FUNCTION_BLOCK IO_RouteAI (* Backend router for IO_AI: 0 simulated, 1 GPIO, 2 Modbus *)
  (* Standard: 61499-2 *)
  (* Version 0.1, 2026-09-28, Project contributors, AAU Smart Production Lab *)
  PACKAGE unitlib;
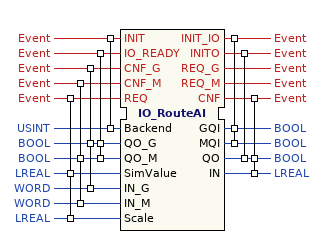
  EVENT_INPUT
    INIT WITH Backend;
    IO_READY WITH QO_G, QO_M;
    CNF_G WITH QO_G, IN_G;
    CNF_M WITH QO_M, IN_M;
    REQ WITH SimValue, Scale;
  END_EVENT
  EVENT_OUTPUT
    INIT_IO WITH GQI, MQI;
    INITO WITH QO;
    REQ_G;
    REQ_M;
    CNF WITH QO, IN;
  END_EVENT
  VAR_INPUT
    Backend : USINT;
    QO_G : BOOL;
    QO_M : BOOL;
    SimValue : LREAL;
    IN_G : WORD;
    IN_M : WORD;
    Scale : LREAL := 1.0;
  END_VAR
  VAR_OUTPUT
    GQI : BOOL;
    MQI : BOOL;
    QO : BOOL;
    IN : LREAL;
  END_VAR
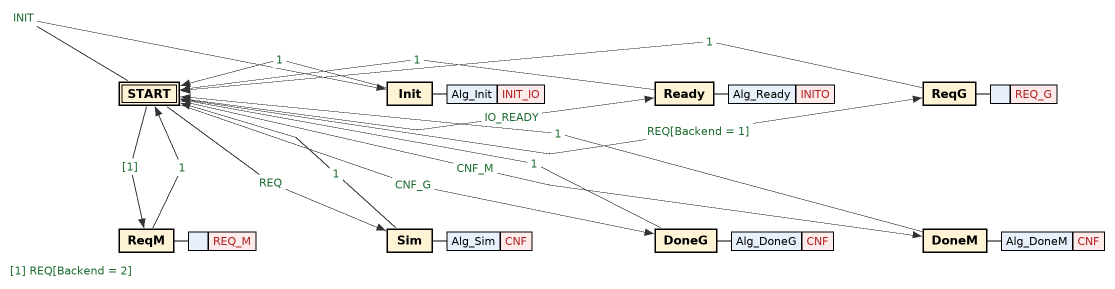
  EC_STATES
    START;
    Init : Alg_Init -> INIT_IO;
    Ready : Alg_Ready -> INITO;
    ReqG : -> REQ_G;
    ReqM : -> REQ_M;
    Sim : Alg_Sim -> CNF;
    DoneG : Alg_DoneG -> CNF;
    DoneM : Alg_DoneM -> CNF;
  END_STATES
  EC_TRANSITIONS
    START TO Init := INIT;
    Init TO START := 1;
    START TO Ready := IO_READY;
    Ready TO START := 1;
    START TO ReqG := REQ[Backend = 1];
    START TO ReqM := REQ[Backend = 2];
    START TO Sim := REQ;
    START TO DoneG := CNF_G;
    START TO DoneM := CNF_M;
    ReqG TO START := 1;
    ReqM TO START := 1;
    Sim TO START := 1;
    DoneG TO START := 1;
    DoneM TO START := 1;
  END_TRANSITIONS
  ALGORITHM Alg_Init IN ST:
GQI := Backend = 1;
MQI := Backend = 2;
  END_ALGORITHM
  ALGORITHM Alg_Ready IN ST:
QO := (Backend = 0) OR ((Backend = 1) AND QO_G) OR ((Backend = 2) AND QO_M);
  END_ALGORITHM
  ALGORITHM Alg_Sim IN ST:
QO := TRUE;
IN := SimValue;
  END_ALGORITHM
  ALGORITHM Alg_DoneG IN ST:
QO := QO_G;
IN := UINT_TO_LREAL(WORD_TO_UINT(IN_G)) * Scale;
  END_ALGORITHM
  ALGORITHM Alg_DoneM IN ST:
QO := QO_M;
IN := UINT_TO_LREAL(WORD_TO_UINT(IN_M)) * Scale;
  END_ALGORITHM
END_FUNCTION_BLOCK
